(* IEC 61131-3 sources: POMIRTS_lab3/AS/Library_2/AsHydCon/V3.00.0, 3 files *)

(* ---- AsHydCon.typ ---- *)
TYPE
	HCRMovePara_typ : STRUCT
		t_Jolt	: REAL ;
		vC_pos	: REAL ;
		vC_neg	: REAL ;
		aAcc_pos	: REAL ;
		aDec_pos	: REAL ;
		aAcc_neg	: REAL ;
		aDec_neg	: REAL ;
	END_STRUCT;
	HCRSFG_Internal_typ : STRUCT
		SFG_Para	: HCRMovePara_typ ;
		Profile_Case	: USINT ;
		Fp_delta	: REAL ;
		Fp_brake	: REAL ;
		Fp_set_0	: REAL ;
		dFp_set_0	: REAL ;
		dFp_home	: REAL ;
		dFp_0_intrude	: USINT ;
		dFp_const	: REAL ;
		dFp_const_avg	: REAL ;
		dFp_thresh	: ARRAY[0..2] OF REAL ;
		t_Jolt	: REAL ;
		t_delta	: REAL ;
		t_delta_Jolt	: REAL ;
		t_delta_3_Jolt	: REAL ;
		Calc_t_delta	: USINT ;
		tx	: REAL ;
		tx_limit	: REAL ;
		enable_old	: BOOL ;
		Bootkey	: UDINT ;
	END_STRUCT;
	HCRF_Cont_InVar_typ : STRUCT
		I_Switch	: USINT ;
		Q_man	: REAL ;
		Q_add	: REAL ;
		v_act	: REAL ;
		Qy_Oset_ext	: REAL ;
		Oset_Mode	: USINT ;
	END_STRUCT;
	HCRP2P_Cont_Internal_typ : STRUCT
		MoveDir	: SINT ;
		s_set_old	: REAL ;
		enable_old	: BOOL ;
		Bootkey	: UDINT ;
	END_STRUCT;
	HCRP2P_Cont_AddPar_typ : STRUCT
		Y_P2P_min	: REAL ;
		Y_P2P_max	: REAL ;
		dY_max	: REAL ;
		Tn_pos	: REAL ;
		Tn_neg	: REAL ;
		I_Switch	: USINT ;
		Tv	: REAL ;
		Tf	: REAL ;
	END_STRUCT;
	HCRF_Cont_p_Internal_typ : STRUCT
		Qnom_pos	: REAL ;
		Qnom_neg	: REAL ;
		Oset_Mode	: USINT ;
		Qy_Oset_F_pos	: REAL ;
		Qy_Oset_F_neg	: REAL ;
		enable_old	: BOOL ;
		Bootkey	: UDINT ;
	END_STRUCT;
	HCRFyServo_Internal_typ : STRUCT
		E	: REAL ;
		Alpha	: REAL ;
		pSupply_max	: REAL ;
		pSupply	: REAL ;
		pTank	: REAL ;
		Qnom_pos	: REAL ;
		Qnom_neg	: REAL ;
		A_Cyl_pos	: REAL ;
		A_Cyl_neg	: REAL ;
		V0_pos	: REAL ;
		V0_neg	: REAL ;
		Neg_y	: BOOL ;
		dF_Cyl_sup	: REAL ;
		dF_Cyl_sum	: REAL ;
		x_Cyl	: REAL ;
		h_Cyl	: REAL ;
		h_Cyl_dbl_1	: UDINT ;
		h_Cyl_dbl_2	: UDINT ;
		K_pos_dbl_1	: UDINT ;
		K_pos_dbl_2	: UDINT ;
		K_neg_dbl_1	: UDINT ;
		K_neg_dbl_2	: UDINT ;
		V0_A_Cyl_pos_dbl_1	: UDINT ;
		V0_A_Cyl_pos_dbl_2	: UDINT ;
		V0_A_Cyl_neg_dbl_1	: UDINT ;
		V0_A_Cyl_neg_dbl_2	: UDINT ;
		A_Cyl_pos_1000_dbl_1	: UDINT ;
		A_Cyl_pos_1000_dbl_2	: UDINT ;
		A_Cyl_neg_1000_dbl_1	: UDINT ;
		A_Cyl_neg_1000_dbl_2	: UDINT ;
		E_10_dbl_1	: UDINT ;
		E_10_dbl_2	: UDINT ;
		pDelta_min_dbl_1	: UDINT ;
		pDelta_min_dbl_2	: UDINT ;
		dF_Cyl_sup_100_dbl_1	: UDINT ;
		dF_Cyl_sup_100_dbl_2	: UDINT ;
		Update_old	: USINT ;
		Update_2	: USINT ;
		enable_old	: BOOL ;
		Bootkey	: UDINT ;
	END_STRUCT;
	HCRNotch_Internal_typ : STRUCT
		Ts	: DINT ;
		Ts_dbl_1	: UDINT ;
		Ts_dbl_2	: UDINT ;
		fs_dbl_1	: UDINT ;
		fs_dbl_2	: UDINT ;
		V_old	: REAL ;
		f0_old	: REAL ;
		B_old	: REAL ;
		Set_y_old	: USINT ;
		Set_y_2	: USINT ;
		fg_upper	: REAL ;
		fg_lower	: REAL ;
		B_act	: REAL ;
		D	: REAL ;
		Tf	: REAL ;
		x1_dbl_1	: UDINT ;
		x1_dbl_2	: UDINT ;
		x2_dbl_1	: UDINT ;
		x2_dbl_2	: UDINT ;
		D_Ts_Tf_dbl_1	: UDINT ;
		D_Ts_Tf_dbl_2	: UDINT ;
		Sqrt_D_1_dbl_1	: UDINT ;
		Sqrt_D_1_dbl_2	: UDINT ;
		a0_dbl_1	: UDINT ;
		a0_dbl_2	: UDINT ;
		a1_dbl_1	: UDINT ;
		a1_dbl_2	: UDINT ;
		b0_dbl_1	: UDINT ;
		b0_dbl_2	: UDINT ;
		b1_dbl_1	: UDINT ;
		b1_dbl_2	: UDINT ;
		Bootkey	: UDINT ;
	END_STRUCT;
	HCRIT1_Internal_typ : STRUCT
		Ts	: DINT ;
		Ts_dbl_1	: UDINT ;
		Ts_dbl_2	: UDINT ;
		V_old	: REAL ;
		Tn_old	: REAL ;
		T1_old	: REAL ;
		Set_y_old	: USINT ;
		Set_y_2	: USINT ;
		x1_dbl_1	: UDINT ;
		x1_dbl_2	: UDINT ;
		x2_dbl_1	: UDINT ;
		x2_dbl_2	: UDINT ;
		Exp_Ts_T1_dbl_1	: UDINT ;
		Exp_Ts_T1_dbl_2	: UDINT ;
		V_Tn_dbl_1	: UDINT ;
		V_Tn_dbl_2	: UDINT ;
		a0_dbl_1	: UDINT ;
		a0_dbl_2	: UDINT ;
		a1_dbl_1	: UDINT ;
		a1_dbl_2	: UDINT ;
		b0_dbl_1	: UDINT ;
		b0_dbl_2	: UDINT ;
		b1_dbl_1	: UDINT ;
		b1_dbl_2	: UDINT ;
		Bootkey	: UDINT ;
	END_STRUCT;
	HCRSystemParaAdd_typ : STRUCT
		V0_pos	: REAL ;
		V0_neg	: REAL ;
		h_Cyl	: REAL ;
		m_Cyl	: REAL ;
	END_STRUCT;
	HCRRampGen_Internal_typ : STRUCT
		t_rise	: REAL ;
		t_hold	: REAL ;
		t_fall	: REAL ;
		y	: REAL ;
		dy	: REAL ;
		Finished	: BOOL ;
		Ts	: DINT ;
		Ts_dbl_1	: UDINT ;
		Ts_dbl_2	: UDINT ;
		Timer_dbl_1	: UDINT ;
		Timer_dbl_2	: UDINT ;
		k_Ramp_dbl_1	: UDINT ;
		k_Ramp_dbl_2	: UDINT ;
		y_dbl_1	: UDINT ;
		y_dbl_2	: UDINT ;
		RampGenPhase	: USINT ;
		enable_old	: BOOL ;
		Bootkey	: UDINT ;
	END_STRUCT;
	HCRAutoTune_Internal_typ : STRUCT
		E	: REAL ;
		V0_pos	: REAL ;
		V0_pos_mod_dbl_1	: UDINT ;
		V0_pos_mod_dbl_2	: UDINT ;
		V0_neg	: REAL ;
		V0_neg_mod_dbl_1	: UDINT ;
		V0_neg_mod_dbl_2	: UDINT ;
		s_Cyl_min_dbl_1	: UDINT ;
		s_Cyl_min_dbl_2	: UDINT ;
		s_Cyl_max_dbl_1	: UDINT ;
		s_Cyl_max_dbl_2	: UDINT ;
		h_Cyl	: REAL ;
		h_Cyl_dbl_1	: UDINT ;
		h_Cyl_dbl_2	: UDINT ;
		E_A_pos_2_dbl_1	: UDINT ;
		E_A_pos_2_dbl_2	: UDINT ;
		E_A_neg_2_dbl_1	: UDINT ;
		E_A_neg_2_dbl_2	: UDINT ;
		s0_Cyl	: REAL ;
		s0_Cyl_dbl_1	: UDINT ;
		s0_Cyl_dbl_2	: UDINT ;
		c0_Cyl	: REAL ;
		c0_Cyl_dbl_1	: UDINT ;
		c0_Cyl_dbl_2	: UDINT ;
		omega0_Cyl	: REAL ;
		omega0_Cyl_dbl_1	: UDINT ;
		omega0_Cyl_dbl_2	: UDINT ;
		vCyl_sup_pos	: REAL ;
		vCyl_sup_neg	: REAL ;
		vCyl_sup	: REAL ;
		Kp_dbl_1	: UDINT ;
		Kp_dbl_2	: UDINT ;
		Kp_physical	: REAL ;
		enable_old	: BOOL ;
		Bootkey	: UDINT ;
	END_STRUCT;
	HCRs_Cont_p_InVar_typ : STRUCT
		I_Switch	: USINT ;
		v_man	: REAL ;
		v_add	: REAL ;
		v_set	: REAL ;
		pCyl_pos	: REAL ;
		pCyl_neg	: REAL ;
		Qy_Oset_ext	: REAL ;
		Oset_Mode	: USINT ;
	END_STRUCT;
	HCRsF_Cont_p_Internal_typ : STRUCT
		CTRLmode	: USINT ;
		uSwitch_old	: USINT ;
		enable_old	: BOOL ;
		Bootkey	: UDINT ;
	END_STRUCT;
	HCRs_Cont_p_Internal_typ : STRUCT
		vCyl_sup_pos	: REAL ;
		vCyl_sup_neg	: REAL ;
		vCyl_sup	: REAL ;
		s_set_old	: REAL ;
		s_act_old	: REAL ;
		v_act	: REAL ;
		Oset_Mode	: USINT ;
		Qy_Oset_s_pos	: REAL ;
		Qy_Oset_s_neg	: REAL ;
		Qy_I_Switch	: USINT ;
		Qy_I	: REAL ;
		MoveDir_I	: SINT ;
		enable_old	: BOOL ;
		Bootkey	: UDINT ;
	END_STRUCT;
	HCROmega0_Internal_typ : STRUCT
		E	: REAL ;
		Kp_xCorr_Lim	: REAL ;
		A_Cyl_pos	: REAL ;
		A_Cyl_neg	: REAL ;
		V0_pos	: REAL ;
		V0_neg	: REAL ;
		h_Cyl	: REAL ;
		x_Cyl_min_dbl_1	: UDINT ;
		x_Cyl_min_dbl_2	: UDINT ;
		x_Cyl_max_dbl_1	: UDINT ;
		x_Cyl_max_dbl_2	: UDINT ;
		E_A_pos_2_dbl_1	: UDINT ;
		E_A_pos_2_dbl_2	: UDINT ;
		E_A_neg_2_dbl_1	: UDINT ;
		E_A_neg_2_dbl_2	: UDINT ;
		x0_Cyl_dbl_1	: UDINT ;
		x0_Cyl_dbl_2	: UDINT ;
		c0_Cyl	: REAL ;
		c0_Cyl_dbl_1	: UDINT ;
		c0_Cyl_dbl_2	: UDINT ;
		c_Cyl_Lim_L	: REAL ;
		c_Cyl_Lim_L_dbl_1	: UDINT ;
		c_Cyl_Lim_L_dbl_2	: UDINT ;
		c_Cyl_Lim_R	: REAL ;
		c_Cyl_Lim_R_dbl_1	: UDINT ;
		c_Cyl_Lim_R_dbl_2	: UDINT ;
		c_Cyl	: REAL ;
		c_Cyl_dbl_1	: UDINT ;
		c_Cyl_dbl_2	: UDINT ;
		Kp_xCorr_Lim_L	: REAL ;
		Kp_xCorr_Lim_R	: REAL ;
		enable_old	: BOOL ;
		Bootkey	: UDINT ;
	END_STRUCT;
	HCRLinValve_Internal_typ : STRUCT
		Neg_Uy	: BOOL ;
		enable_old	: BOOL ;
		Bootkey	: UDINT ;
	END_STRUCT;
	HCRFIFO_Internal_typ : STRUCT
		Ts	: DINT ;
		t_FIFO_max	: DINT ;
		MemSize	: UDINT ;
		MemSize_REAL	: UDINT ;
		Set_y_2	: BOOL ;
		pFIFO_Buf	: UDINT ;
		pFIFO_OutIn	: UDINT ;
		enable_old	: BOOL ;
		Bootkey	: UDINT ;
	END_STRUCT;
	HCRDT2_Internal_typ : STRUCT
		Ts	: DINT ;
		Ts_dbl_1	: UDINT ;
		Ts_dbl_2	: UDINT ;
		Tv_old	: REAL ;
		T1_old	: REAL ;
		T2_old	: REAL ;
		n_Avg_old	: USINT ;
		u_Buf	: ARRAY[0..99] OF REAL ;
		u_BufCnt	: SINT ;
		u_Sum_dbl_1	: UDINT ;
		u_Sum_dbl_2	: UDINT ;
		u_Avg_dbl_1	: UDINT ;
		u_Avg_dbl_2	: UDINT ;
		Reset_y_old	: USINT ;
		Reset_y_2	: USINT ;
		x1_dbl_1	: UDINT ;
		x1_dbl_2	: UDINT ;
		x2_dbl_1	: UDINT ;
		x2_dbl_2	: UDINT ;
		Tv_T1_dbl_1	: UDINT ;
		Tv_T1_dbl_2	: UDINT ;
		Tv_T2_dbl_1	: UDINT ;
		Tv_T2_dbl_2	: UDINT ;
		Exp_Ts_T1_dbl_1	: UDINT ;
		Exp_Ts_T1_dbl_2	: UDINT ;
		Exp_Ts_T2_dbl_1	: UDINT ;
		Exp_Ts_T2_dbl_2	: UDINT ;
		Exp_T1_T2_dbl_1	: UDINT ;
		Exp_T1_T2_dbl_2	: UDINT ;
		a0_dbl_1	: UDINT ;
		a0_dbl_2	: UDINT ;
		a1_dbl_1	: UDINT ;
		a1_dbl_2	: UDINT ;
		b0_dbl_1	: UDINT ;
		b0_dbl_2	: UDINT ;
		b1_dbl_1	: UDINT ;
		b1_dbl_2	: UDINT ;
		Bootkey	: UDINT ;
	END_STRUCT;
	HCRF_Cont_p_InVar_typ : STRUCT
		I_Switch	: USINT ;
		Q_man	: REAL ;
		Q_add	: REAL ;
		dFp_set	: REAL ;
		x_Cyl	: REAL ;
		v_Cyl	: REAL ;
		pCyl_pos	: REAL ;
		pCyl_neg	: REAL ;
		v_act	: REAL ;
		Qy_Oset_ext	: REAL ;
		Oset_Mode	: USINT ;
	END_STRUCT;
	HCRs_Cont_InVar_typ : STRUCT
		I_Switch	: USINT ;
		v_man	: REAL ;
		v_add	: REAL ;
		v_set	: REAL ;
		Fp_Cyl	: REAL ;
		Ff_Cyl_pos	: REAL ;
		Ff_Cyl_neg	: REAL ;
		Qy_Oset_ext	: REAL ;
		Oset_Mode	: USINT ;
	END_STRUCT;
	HCRsF_Cont_Internal_typ : STRUCT
		uSwitch_old	: USINT ;
		enable_old	: BOOL ;
		Bootkey	: UDINT ;
	END_STRUCT;
	HCRPIDPara_F_typ : STRUCT
		Fp_min	: REAL ;
		Fp_max	: REAL ;
		Kw	: REAL ;
		Kp	: REAL ;
		Tn	: REAL ;
		K_Fbk	: REAL ;
		d_mode	: USINT ;
		Tv	: REAL ;
		Tf	: REAL ;
		dQ_max	: REAL ;
		Q_min	: REAL ;
		Q_max	: REAL ;
	END_STRUCT;
	HCRPIDPara_s_typ : STRUCT
		s_min	: REAL ;
		s_max	: REAL ;
		Kw	: REAL ;
		Kp	: REAL ;
		Tn_pos	: REAL ;
		Tn_neg	: REAL ;
		K_Fbk	: REAL ;
		d_mode	: USINT ;
		Tv	: REAL ;
		Tf	: REAL ;
		dv_max	: REAL ;
		v_min	: REAL ;
		v_max	: REAL ;
	END_STRUCT;
	HCRF_Cont_Internal_typ : STRUCT
		Qnom_pos	: REAL ;
		Qnom_neg	: REAL ;
		Oset_Mode	: USINT ;
		Qy_Oset_F_pos	: REAL ;
		Qy_Oset_F_neg	: REAL ;
		enable_old	: BOOL ;
		Bootkey	: UDINT ;
	END_STRUCT;
	HCRJoltFree_Internal_typ : STRUCT
		uSwitch_old	: BOOL ;
		enable_old	: BOOL ;
		Bootkey	: UDINT ;
	END_STRUCT;
	HCRDT2s_Internal_typ : STRUCT
		Ts	: DINT ;
		Ts_dbl_1	: UDINT ;
		Ts_dbl_2	: UDINT ;
		D_old	: REAL ;
		Tv_old	: REAL ;
		Tf_old	: REAL ;
		Reset_y_old	: USINT ;
		Reset_y_2	: USINT ;
		x1_dbl_1	: UDINT ;
		x1_dbl_2	: UDINT ;
		x2_dbl_1	: UDINT ;
		x2_dbl_2	: UDINT ;
		Sqrt_D_1_dbl_1	: UDINT ;
		Sqrt_D_1_dbl_2	: UDINT ;
		Tv_Tf_dbl_1	: UDINT ;
		Tv_Tf_dbl_2	: UDINT ;
		Ts_Tf_dbl_1	: UDINT ;
		Ts_Tf_dbl_2	: UDINT ;
		Exp_D_Ts_Tf_dbl_1	: UDINT ;
		Exp_D_Ts_Tf_dbl_2	: UDINT ;
		a0_dbl_1	: UDINT ;
		a0_dbl_2	: UDINT ;
		a1_dbl_1	: UDINT ;
		a1_dbl_2	: UDINT ;
		b0_dbl_1	: UDINT ;
		b0_dbl_2	: UDINT ;
		b1_dbl_1	: UDINT ;
		b1_dbl_2	: UDINT ;
		Bootkey	: UDINT ;
	END_STRUCT;
	HCRPT1cP_Internal_typ : STRUCT
		Ts	: DINT ;
		Ts_dbl_1	: UDINT ;
		Ts_dbl_2	: UDINT ;
		T1_intern	: REAL ;
		nCnt	: UDINT ;
		Set_y_old	: USINT ;
		Set_y_2	: USINT ;
		x_dbl_1	: UDINT ;
		x_dbl_2	: UDINT ;
		Exp_5_dbl_1	: UDINT ;
		Exp_5_dbl_2	: UDINT ;
		a0_dbl_1	: UDINT ;
		a0_dbl_2	: UDINT ;
		b0_dbl_1	: UDINT ;
		b0_dbl_2	: UDINT ;
		Bootkey	: UDINT ;
	END_STRUCT;
	HCRPT2s_Internal_typ : STRUCT
		Ts	: DINT ;
		Ts_dbl_1	: UDINT ;
		Ts_dbl_2	: UDINT ;
		V_old	: REAL ;
		D_old	: REAL ;
		Tf_old	: REAL ;
		Set_y_old	: USINT ;
		Set_y_2	: USINT ;
		x1_dbl_1	: UDINT ;
		x1_dbl_2	: UDINT ;
		x2_dbl_1	: UDINT ;
		x2_dbl_2	: UDINT ;
		Sqrt_D_1_dbl_1	: UDINT ;
		Sqrt_D_1_dbl_2	: UDINT ;
		Ts_Tf_dbl_1	: UDINT ;
		Ts_Tf_dbl_2	: UDINT ;
		Exp_D_Ts_Tf_dbl_1	: UDINT ;
		Exp_D_Ts_Tf_dbl_2	: UDINT ;
		a0_dbl_1	: UDINT ;
		a0_dbl_2	: UDINT ;
		a1_dbl_1	: UDINT ;
		a1_dbl_2	: UDINT ;
		b0_dbl_1	: UDINT ;
		b0_dbl_2	: UDINT ;
		b1_dbl_1	: UDINT ;
		b1_dbl_2	: UDINT ;
		Bootkey	: UDINT ;
	END_STRUCT;
	HCRPT2_Internal_typ : STRUCT
		Ts	: DINT ;
		Ts_dbl_1	: UDINT ;
		Ts_dbl_2	: UDINT ;
		V_old	: REAL ;
		T1_old	: REAL ;
		T2_old	: REAL ;
		Set_y_old	: USINT ;
		Set_y_2	: USINT ;
		x1_dbl_1	: UDINT ;
		x1_dbl_2	: UDINT ;
		x2_dbl_1	: UDINT ;
		x2_dbl_2	: UDINT ;
		Exp_Ts_T1_dbl_1	: UDINT ;
		Exp_Ts_T1_dbl_2	: UDINT ;
		Exp_Ts_T2_dbl_1	: UDINT ;
		Exp_Ts_T2_dbl_2	: UDINT ;
		Exp_Ts_T1_T2_dbl_1	: UDINT ;
		Exp_Ts_T1_T2_dbl_2	: UDINT ;
		Exp_T1_T2_dbl_1	: UDINT ;
		Exp_T1_T2_dbl_2	: UDINT ;
		V1_Exp_dbl_1	: UDINT ;
		V1_Exp_dbl_2	: UDINT ;
		V2_Exp_dbl_1	: UDINT ;
		V2_Exp_dbl_2	: UDINT ;
		Bootkey	: UDINT ;
	END_STRUCT;
	HCRPT1_Internal_typ : STRUCT
		Ts	: DINT ;
		Ts_dbl_1	: UDINT ;
		Ts_dbl_2	: UDINT ;
		V_old	: REAL ;
		T1_old	: REAL ;
		Set_y_old	: USINT ;
		Set_y_2	: USINT ;
		x_dbl_1	: UDINT ;
		x_dbl_2	: UDINT ;
		Exp_Ts_T1_dbl_1	: UDINT ;
		Exp_Ts_T1_dbl_2	: UDINT ;
		V_Exp_dbl_1	: UDINT ;
		V_Exp_dbl_2	: UDINT ;
		Bootkey	: UDINT ;
	END_STRUCT;
	HCRDT1_Internal_typ : STRUCT
		Ts	: DINT ;
		Ts_dbl_1	: UDINT ;
		Ts_dbl_2	: UDINT ;
		Tv_old	: REAL ;
		Tf_old	: REAL ;
		n_Avg_old	: USINT ;
		u_Buf	: ARRAY[0..99] OF REAL ;
		u_BufCnt	: SINT ;
		u_Sum_dbl_1	: UDINT ;
		u_Sum_dbl_2	: UDINT ;
		u_Avg_dbl_1	: UDINT ;
		u_Avg_dbl_2	: UDINT ;
		Reset_y_old	: USINT ;
		Reset_y_2	: USINT ;
		x_dbl_1	: UDINT ;
		x_dbl_2	: UDINT ;
		Tv_Tf_dbl_1	: UDINT ;
		Tv_Tf_dbl_2	: UDINT ;
		Exp_Ts_Tf_dbl_1	: UDINT ;
		Exp_Ts_Tf_dbl_2	: UDINT ;
		Tv_Tf_Exp_dbl_1	: UDINT ;
		Tv_Tf_Exp_dbl_2	: UDINT ;
		V_Exp_dbl_1	: UDINT ;
		V_Exp_dbl_2	: UDINT ;
		Bootkey	: UDINT ;
	END_STRUCT;
	HCRFyServo_Fp_Internal_typ : STRUCT
		Alpha	: REAL ;
		pSupply_max	: REAL ;
		pSupply	: REAL ;
		pTank	: REAL ;
		Qnom_pos	: REAL ;
		Qnom_neg	: REAL ;
		A_Cyl_pos	: REAL ;
		A_Cyl_neg	: REAL ;
		Neg_y	: BOOL ;
		Supply_Tank_pos_dbl_1	: UDINT ;
		Supply_Tank_pos_dbl_2	: UDINT ;
		Supply_Tank_neg_dbl_1	: UDINT ;
		Supply_Tank_neg_dbl_2	: UDINT ;
		K_numer_dbl_1	: UDINT ;
		K_numer_dbl_2	: UDINT ;
		Update_old	: USINT ;
		Update_2	: USINT ;
		enable_old	: BOOL ;
		Bootkey	: UDINT ;
	END_STRUCT;
	HCRSPF_Internal_typ : STRUCT
		Profile_Nb	: USINT ;
		Profile_ID	: USINT ;
		Profile_Case	: USINT ;
		MovementPhase	: USINT ;
		MovementStep	: USINT ;
		s_end	: REAL ;
		s_set_0_dbl_1	: UDINT ;
		s_set_0_dbl_2	: UDINT ;
		v_set_0_dbl_1	: UDINT ;
		v_set_0_dbl_2	: UDINT ;
		a_set_0_dbl_1	: UDINT ;
		a_set_0_dbl_2	: UDINT ;
		v0	: REAL ;
		v0_dbl_1	: UDINT ;
		v0_dbl_2	: UDINT ;
		v0_intrude	: USINT ;
		v0_state	: USINT ;
		s_set	: REAL ;
		s_set_Jolt	: REAL ;
		s_set_dbl_1	: UDINT ;
		s_set_dbl_2	: UDINT ;
		v_set	: REAL ;
		v_set_Jolt	: REAL ;
		v_set_dbl_1	: UDINT ;
		v_set_dbl_2	: UDINT ;
		a_set	: REAL ;
		a_set_Jolt	: REAL ;
		a_set_dbl_1	: UDINT ;
		a_set_dbl_2	: UDINT ;
		vC_pos_dbl_1	: UDINT ;
		vC_pos_dbl_2	: UDINT ;
		vC_neg_dbl_1	: UDINT ;
		vC_neg_dbl_2	: UDINT ;
		aAcc_pos_dbl_1	: UDINT ;
		aAcc_pos_dbl_2	: UDINT ;
		aDec_pos_dbl_1	: UDINT ;
		aDec_pos_dbl_2	: UDINT ;
		aAcc_neg_dbl_1	: UDINT ;
		aAcc_neg_dbl_2	: UDINT ;
		aDec_neg_dbl_1	: UDINT ;
		aDec_neg_dbl_2	: UDINT ;
		aDec	: REAL ;
		aDec_intrude	: BOOL ;
		s_period	: REAL ;
		s_period_Sum_dbl_1	: UDINT ;
		s_period_Sum_dbl_2	: UDINT ;
		Nb_period	: DINT ;
		t_Jolt_max	: REAL ;
		t_Jolt_limit	: REAL ;
		t_Jolt	: REAL ;
		t_Jolt_dbl_1	: UDINT ;
		t_Jolt_dbl_2	: UDINT ;
		sDelta	: REAL ;
		sDelta_dbl_1	: UDINT ;
		sDelta_dbl_2	: UDINT ;
		sBrake	: REAL ;
		sBrake_dbl_1	: UDINT ;
		sBrake_dbl_2	: UDINT ;
		vTop	: REAL ;
		vTop_dbl_1	: UDINT ;
		vTop_dbl_2	: UDINT ;
		AccVec_dbl	: ARRAY[0..39] OF UDINT ;
		ConstVec_dbl	: ARRAY[0..39] OF UDINT ;
		DecVec_dbl	: ARRAY[0..39] OF UDINT ;
		AccVec	: ARRAY[0..19] OF REAL ;
		ConstVec	: ARRAY[0..19] OF REAL ;
		DecVec	: ARRAY[0..19] OF REAL ;
		pBuf_s_set	: UDINT ;
		pBuf_v_set	: UDINT ;
		pBuf_a_set	: UDINT ;
		BufCntMax	: DINT ;
		BufCnt	: DINT ;
		BufCnt_t_Jolt	: DINT ;
		Cnt_t_Jolt	: DINT ;
		s_set_Sum_dbl_1	: UDINT ;
		s_set_Sum_dbl_2	: UDINT ;
		D	: REAL ;
		omega0	: REAL ;
		t_pred	: REAL ;
		Ts	: DINT ;
		Ts_dbl_1	: UDINT ;
		Ts_dbl_2	: UDINT ;
		Ts_2_dbl_1	: UDINT ;
		Ts_2_dbl_2	: UDINT ;
		Ts_4_dbl_1	: UDINT ;
		Ts_4_dbl_2	: UDINT ;
		Timer	: REAL ;
		Timer_dbl_1	: UDINT ;
		Timer_dbl_2	: UDINT ;
		Timer_Ts	: REAL ;
		Timer_Ts_dbl_1	: UDINT ;
		Timer_Ts_dbl_2	: UDINT ;
		T_cycle	: REAL ;
		T_cycle_dbl_1	: UDINT ;
		T_cycle_dbl_2	: UDINT ;
		Const_T_cycle	: BOOL ;
		CounterState	: UINT ;
		musecs_old	: UDINT ;
		SysTicks_old	: UDINT ;
		enable_old	: BOOL ;
		Bootkey_T	: UDINT ;
		Bootkey	: UDINT ;
		s_period_ext	: REAL ;
		PeriodicMode_ext	: INT ;
		NewPeriod_ext_out	: SINT ;
	END_STRUCT;
	HCRs_Cont_Internal_typ : STRUCT
		vCyl_sup_pos	: REAL ;
		vCyl_sup_neg	: REAL ;
		vCyl_sup	: REAL ;
		s_set_old	: REAL ;
		s_act_old	: REAL ;
		v_act	: REAL ;
		Oset_Mode	: USINT ;
		Qy_Oset_s_pos	: REAL ;
		Qy_Oset_s_neg	: REAL ;
		Qy_I_Switch	: USINT ;
		Qy_I	: REAL ;
		MoveDir_I	: SINT ;
		enable_old	: BOOL ;
		Bootkey	: UDINT ;
	END_STRUCT;
	HCRSystemPara_typ : STRUCT
		pSupply_max	: REAL ;
		pSupply	: REAL ;
		pTank	: REAL ;
		A_Cyl_pos	: REAL ;
		A_Cyl_neg	: REAL ;
	END_STRUCT;
	HCRValvePara_typ : STRUCT
		Qnom_pos	: REAL ;
		Qnom_neg	: REAL ;
		pDelta_nom	: REAL ;
		yValve_0	: REAL ;
		Neg_y	: BOOL ;
	END_STRUCT;
	HCRPIDPara_typ : STRUCT
		WX_min	: REAL ;
		WX_max	: REAL ;
		Kw	: REAL ;
		Kp	: REAL ;
		Tn_pos	: REAL ;
		Tn_neg	: REAL ;
		K_Fbk	: REAL ;
		d_mode	: USINT ;
		Tv	: REAL ;
		Tf	: REAL ;
		dY_max	: REAL ;
		Y_min	: REAL ;
		Y_max	: REAL ;
	END_STRUCT;
	HCRPID_Internal_typ : STRUCT
		WX_min	: REAL ;
		WX_max	: REAL ;
		_100_WX_delta_dbl_1	: UDINT ;
		_100_WX_delta_dbl_2	: UDINT ;
		W_norm_dbl_1	: UDINT ;
		W_norm_dbl_2	: UDINT ;
		X_norm_dbl_1	: UDINT ;
		X_norm_dbl_2	: UDINT ;
		Invert	: BOOL ;
		e_norm_dbl_1	: UDINT ;
		e_norm_dbl_2	: UDINT ;
		Kp	: REAL ;
		Kw	: REAL ;
		Kp_Kw_1_dbl_1	: UDINT ;
		Kp_Kw_1_dbl_2	: UDINT ;
		Kp_intrude	: REAL ;
		P_intrude	: BOOL ;
		Yp_dbl_1	: UDINT ;
		Yp_dbl_2	: UDINT ;
		Ts	: DINT ;
		Ts_dbl_1	: UDINT ;
		Ts_dbl_2	: UDINT ;
		Tn_pos_dbl_1	: UDINT ;
		Tn_pos_dbl_2	: UDINT ;
		Tn_neg_dbl_1	: UDINT ;
		Tn_neg_dbl_2	: UDINT ;
		Kp_Ts_Tn_pos_dbl_1	: UDINT ;
		Kp_Ts_Tn_pos_dbl_2	: UDINT ;
		Kp_Ts_Tn_neg_dbl_1	: UDINT ;
		Kp_Ts_Tn_neg_dbl_2	: UDINT ;
		Yi_load	: REAL ;
		I_load	: SINT ;
		Yi_dbl_1	: UDINT ;
		Yi_dbl_2	: UDINT ;
		Yi_pos_last_dbl_1	: UDINT ;
		Yi_pos_last_dbl_2	: UDINT ;
		Yi_neg_last_dbl_1	: UDINT ;
		Yi_neg_last_dbl_2	: UDINT ;
		I_Switch_Sign	: SINT ;
		I_Switch	: SINT ;
		I_Switch_old	: SINT ;
		I_Switch_off	: SINT ;
		d_mode	: USINT ;
		D	: REAL ;
		Tv_dbl_1	: UDINT ;
		Tv_dbl_2	: UDINT ;
		Tf_dbl_1	: UDINT ;
		Tf_dbl_2	: UDINT ;
		x1d_dbl_1	: UDINT ;
		x1d_dbl_2	: UDINT ;
		x2d_dbl_1	: UDINT ;
		x2d_dbl_2	: UDINT ;
		a0d_dbl_1	: UDINT ;
		a0d_dbl_2	: UDINT ;
		a1d_dbl_1	: UDINT ;
		a1d_dbl_2	: UDINT ;
		b0d_dbl_1	: UDINT ;
		b0d_dbl_2	: UDINT ;
		b1d_dbl_1	: UDINT ;
		b1d_dbl_2	: UDINT ;
		Yd_dbl_1	: UDINT ;
		Yd_dbl_2	: UDINT ;
		Reset_Yd	: USINT ;
		Y_min	: REAL ;
		Y_max	: REAL ;
		Ytotal_dbl_1	: UDINT ;
		Ytotal_dbl_2	: UDINT ;
		Ylim_dbl_1	: UDINT ;
		Ylim_dbl_2	: UDINT ;
		Y_Fbk_ext	: REAL ;
		Fbk_mode	: USINT ;
		K_Fbk_Kp_dbl_1	: UDINT ;
		K_Fbk_Kp_dbl_2	: UDINT ;
		e_Fbk_dbl_1	: UDINT ;
		e_Fbk_dbl_2	: UDINT ;
		dY_max	: REAL ;
		dY_max_Ts_dbl_1	: UDINT ;
		dY_max_Ts_dbl_2	: UDINT ;
		Y_dbl_1	: UDINT ;
		Y_dbl_2	: UDINT ;
		UpdateValid	: BOOL ;
		enable_old	: BOOL ;
		Bootkey_CM	: UDINT ;
		Bootkey	: UDINT ;
	END_STRUCT;
	HCRvyServo_Internal_typ : STRUCT
		Alpha	: REAL ;
		vCyl_sup_pos	: REAL ;
		vCyl_sup_neg	: REAL ;
		vCyl_sup	: REAL ;
		vCyl_max_pos	: REAL ;
		vCyl_max_neg	: REAL ;
		vCyl_max	: REAL ;
		vCyl_sum	: REAL ;
		vCyl_thresh	: REAL ;
		vCyl_nOverlap_pos	: REAL ;
		vCyl_nOverlap_neg	: REAL ;
		vCyl_old	: REAL ;
		pSupply_max	: REAL ;
		pSupply	: REAL ;
		pTank	: REAL ;
		Qnom_pos	: REAL ;
		Qnom_neg	: REAL ;
		A_Cyl_pos	: REAL ;
		A_Cyl_neg	: REAL ;
		yValve_zero	: REAL ;
		yValve_min	: REAL ;
		Neg_y	: BOOL ;
		yValve_0	: REAL ;
		yValve_0_dbl_1	: UDINT ;
		yValve_0_dbl_2	: UDINT ;
		K_pos_dbl_1	: UDINT ;
		K_pos_dbl_2	: UDINT ;
		K_neg_dbl_1	: UDINT ;
		K_neg_dbl_2	: UDINT ;
		K_nOverlap_pos_dbl_1	: UDINT ;
		K_nOverlap_pos_dbl_2	: UDINT ;
		K_nOverlap_neg_dbl_1	: UDINT ;
		K_nOverlap_neg_dbl_2	: UDINT ;
		S_nOverlap_dbl_1	: UDINT ;
		S_nOverlap_dbl_2	: UDINT ;
		pDelta_min_dbl_1	: UDINT ;
		pDelta_min_dbl_2	: UDINT ;
		vCyl_sup_100_dbl_1	: UDINT ;
		vCyl_sup_100_dbl_2	: UDINT ;
		Update_old	: USINT ;
		Update_2	: USINT ;
		enable_old	: BOOL ;
		Bootkey	: UDINT ;
	END_STRUCT;
	HCRvyServo_Fp_Internal_typ : STRUCT
		Alpha	: REAL ;
		vCyl_sup_pos	: REAL ;
		vCyl_sup_neg	: REAL ;
		vCyl_sup	: REAL ;
		vCyl_max_pos	: REAL ;
		vCyl_max_neg	: REAL ;
		vCyl_max	: REAL ;
		vCyl_sum	: REAL ;
		vCyl_thresh	: REAL ;
		vCyl_nOverlap_pos	: REAL ;
		vCyl_nOverlap_neg	: REAL ;
		vCyl_old	: REAL ;
		pSupply_max	: REAL ;
		pSupply	: REAL ;
		pTank	: REAL ;
		Qnom_pos	: REAL ;
		Qnom_neg	: REAL ;
		A_Cyl_pos	: REAL ;
		A_Cyl_neg	: REAL ;
		pCyl_pos	: REAL ;
		pCyl_neg	: REAL ;
		yValve_zero	: REAL ;
		yValve_min	: REAL ;
		Neg_y	: BOOL ;
		yValve_0	: REAL ;
		yValve_0_dbl_1	: UDINT ;
		yValve_0_dbl_2	: UDINT ;
		Supply_Tank_pos_dbl_1	: UDINT ;
		Supply_Tank_pos_dbl_2	: UDINT ;
		Supply_Tank_neg_dbl_1	: UDINT ;
		Supply_Tank_neg_dbl_2	: UDINT ;
		Qn_pos_2_A_neg_2_dbl_1	: UDINT ;
		Qn_pos_2_A_neg_2_dbl_2	: UDINT ;
		Qn_neg_2_A_pos_2_dbl_1	: UDINT ;
		Qn_neg_2_A_pos_2_dbl_2	: UDINT ;
		Qn_pos_2_A_neg_3_dbl_1	: UDINT ;
		Qn_pos_2_A_neg_3_dbl_2	: UDINT ;
		Qn_neg_2_A_pos_3_dbl_1	: UDINT ;
		Qn_neg_2_A_pos_3_dbl_2	: UDINT ;
		K_dbl_1	: UDINT ;
		K_dbl_2	: UDINT ;
		K_pos_dbl_1	: UDINT ;
		K_pos_dbl_2	: UDINT ;
		K_neg_dbl_1	: UDINT ;
		K_neg_dbl_2	: UDINT ;
		K_nOverlap_dbl_1	: UDINT ;
		K_nOverlap_dbl_2	: UDINT ;
		K_nOverlap_pos_dbl_1	: UDINT ;
		K_nOverlap_pos_dbl_2	: UDINT ;
		K_nOverlap_neg_dbl_1	: UDINT ;
		K_nOverlap_neg_dbl_2	: UDINT ;
		S_nOverlap_dbl_1	: UDINT ;
		S_nOverlap_dbl_2	: UDINT ;
		pCyl_pos_Numer_pos_dbl_1	: UDINT ;
		pCyl_pos_Numer_pos_dbl_2	: UDINT ;
		pCyl_neg_Numer_pos_dbl_1	: UDINT ;
		pCyl_neg_Numer_pos_dbl_2	: UDINT ;
		pCyl_pos_Numer_neg_dbl_1	: UDINT ;
		pCyl_pos_Numer_neg_dbl_2	: UDINT ;
		pCyl_neg_Numer_neg_dbl_1	: UDINT ;
		pCyl_neg_Numer_neg_dbl_2	: UDINT ;
		pCyl_Denom_dbl_1	: UDINT ;
		pCyl_Denom_dbl_2	: UDINT ;
		vCyl_sup_100_dbl_1	: UDINT ;
		vCyl_sup_100_dbl_2	: UDINT ;
		Update_old	: USINT ;
		Update_2	: USINT ;
		enable_old	: BOOL ;
		Bootkey	: UDINT ;
	END_STRUCT;
	HCRLinSpline_Internal_typ : STRUCT
		AscendingX_o	: SINT ;
		AscendingXs_o	: SINT ;
		AscendingY_o	: SINT ;
		AscendingYs_o	: SINT ;
		AscendingX_d	: SINT ;
		AscendingXs_d	: SINT ;
		AscendingY_d	: SINT ;
		AscendingYs_d	: SINT ;
		Rness_crit	: REAL ;
		RnessP	: REAL ;
		RnessR	: REAL ;
		_Smooth1_dbl_1	: UDINT ;
		_Smooth1_dbl_2	: UDINT ;
		_1Smooth_dbl_1	: UDINT ;
		_1Smooth_dbl_2	: UDINT ;
		_1Smooth1_dbl_1	: UDINT ;
		_1Smooth1_dbl_2	: UDINT ;
		enable_old	: BOOL ;
		Bootkey	: UDINT ;
	END_STRUCT;
	HCRNode_Internal_typ : STRUCT
		X	: REAL ;
		Y	: REAL ;
		X1	: REAL ;
		X2	: REAL ;
		Rness_crit	: REAL ;
		X1_dbl_1	: UDINT ;
		X1_dbl_2	: UDINT ;
		X2_dbl_1	: UDINT ;
		X2_dbl_2	: UDINT ;
		deltaX_dbl_1	: UDINT ;
		deltaX_dbl_2	: UDINT ;
		deltaY_dbl_1	: UDINT ;
		deltaY_dbl_2	: UDINT ;
		k_dbl_1	: UDINT ;
		k_dbl_2	: UDINT ;
		d_dbl_1	: UDINT ;
		d_dbl_2	: UDINT ;
	END_STRUCT;
	HCRNode_typ : STRUCT
		X	: REAL ;
		Y	: REAL ;
		Internal	: HCRNode_Internal_typ ;
	END_STRUCT;
END_TYPE

(* ---- AsHydCon.fun ---- *)
FUNCTION_BLOCK HCRsF_Cont_p (* Switchable position/force controller (pressure). *)
	VAR_INPUT
		enable	:BOOL;
		pSystem_Para	:REFERENCE TO HCRSystemPara_typ;
		pSystem_ParaAdd	:REFERENCE TO HCRSystemParaAdd_typ;
		pValve_Para	:REFERENCE TO HCRValvePara_typ;
		pPID_Para_s	:REFERENCE TO HCRPIDPara_s_typ;
		pPID_Para_F	:REFERENCE TO HCRPIDPara_F_typ;
		vyServoMode	:USINT;
		FyServoMode	:USINT;
		tSwitch	:REAL;
		Update	:USINT;
		s_set	:REAL;
		s_act	:REAL;
		s_Cont_p_InVar	:HCRs_Cont_p_InVar_typ;
		Fp_set	:REAL;
		Fp_act	:REAL;
		F_Cont_InVar	:HCRF_Cont_p_InVar_typ;
		CTRLmode	:USINT;
		uSwitch	:USINT;
	END_VAR
	VAR_OUTPUT
		Qy_s	:REAL;
		Qy_Oset_s	:REAL;
		Qy_F	:REAL;
		Qy_Oset_F	:REAL;
		Qy	:REAL;
		yValve	:REAL;
		MoveDir	:SINT;
		status	:UINT;
	END_VAR
	VAR
		Internal	:HCRsF_Cont_p_Internal_typ;
		s_Cont_p	:HCRs_Cont_p;
		F_Cont	:HCRF_Cont;
		F_Cont_p	:HCRF_Cont_p;
		vyServo	:HCRvyServo;
		JoltFree	:HCRJoltFree;
	END_VAR
END_FUNCTION_BLOCK
FUNCTION_BLOCK HCRNotch (* 2nd order notch filter. *)
	VAR_INPUT
		enable	:BOOL;
		V	:REAL;
		f0	:REAL;
		B	:REAL;
		u	:REAL;
		Set_y	:USINT;
		y_set	:REAL;
	END_VAR
	VAR_OUTPUT
		y	:REAL;
		status	:UINT;
	END_VAR
	VAR
		Internal	:HCRNotch_Internal_typ;
	END_VAR
END_FUNCTION_BLOCK
FUNCTION_BLOCK HCRs_Cont_p (* Position controller (pressure). *)
	VAR_INPUT
		enable	:BOOL;
		pSystem_Para	:REFERENCE TO HCRSystemPara_typ;
		pValve_Para	:REFERENCE TO HCRValvePara_typ;
		pPID_Para_s	:REFERENCE TO HCRPIDPara_s_typ;
		vyServoMode	:USINT;
		Update	:USINT;
		s_set	:REAL;
		s_act	:REAL;
		Invert	:BOOL;
		I_Switch	:USINT;
		CTRLmode	:USINT;
		v_man	:REAL;
		v_add	:REAL;
		v_set	:REAL;
		pCyl_pos	:REAL;
		pCyl_neg	:REAL;
		Qy_Oset_ext	:REAL;
		Oset_Mode	:USINT;
	END_VAR
	VAR_OUTPUT
		Qy_s	:REAL;
		Qy_Oset_s	:REAL;
		Qy	:REAL;
		yValve	:REAL;
		MoveDir	:SINT;
		status	:UINT;
	END_VAR
	VAR
		Internal	:HCRs_Cont_p_Internal_typ;
		PID	:HCRPID;
		vyServo	:HCRvyServo;
	END_VAR
END_FUNCTION_BLOCK
FUNCTION_BLOCK HCRAutoTune (* Autotuning-algorithm for Kp. *)
	VAR_INPUT
		enable	:BOOL;
		pSupply_max	:REAL;
		A_Cyl_pos	:REAL;
		A_Cyl_neg	:REAL;
		Qnom_pos	:REAL;
		Qnom_neg	:REAL;
		pDelta_nom	:REAL;
		V0_pos	:REAL;
		V0_neg	:REAL;
		h_Cyl	:REAL;
		m_Cyl	:REAL;
		s_min	:REAL;
		s_max	:REAL;
		Update	:USINT;
	END_VAR
	VAR_OUTPUT
		Kp	:REAL;
		status	:UINT;
	END_VAR
	VAR
		Internal	:HCRAutoTune_Internal_typ;
	END_VAR
END_FUNCTION_BLOCK
FUNCTION_BLOCK HCRRampGen (* Ramp generator. *)
	VAR_INPUT
		enable	:BOOL;
		t_rise	:REAL;
		t_hold	:REAL;
		t_fall	:REAL;
		y_start	:REAL;
		y_hold	:REAL;
		y_end	:REAL;
		Init	:BOOL;
	END_VAR
	VAR_OUTPUT
		y	:REAL;
		dy	:REAL;
		Finished	:BOOL;
		status	:UINT;
	END_VAR
	VAR
		Internal	:HCRRampGen_Internal_typ;
	END_VAR
END_FUNCTION_BLOCK
FUNCTION_BLOCK HCRPT1 (* 1st order delay element. *)
	VAR_INPUT
		enable	:BOOL;
		V	:REAL;
		T1	:REAL;
		u	:REAL;
		Set_y	:USINT;
		y_set	:REAL;
	END_VAR
	VAR_OUTPUT
		y	:REAL;
		status	:UINT;
	END_VAR
	VAR
		Internal	:HCRPT1_Internal_typ;
	END_VAR
END_FUNCTION_BLOCK
FUNCTION_BLOCK HCRDT1 (* 1st order differentiator. *)
	VAR_INPUT
		enable	:BOOL;
		Tv	:REAL;
		Tf	:REAL;
		u	:REAL;
		n_Avg	:USINT;
		Reset_y	:USINT;
	END_VAR
	VAR_OUTPUT
		y	:REAL;
		status	:UINT;
	END_VAR
	VAR
		Internal	:HCRDT1_Internal_typ;
	END_VAR
END_FUNCTION_BLOCK
FUNCTION_BLOCK HCRLinSpline (* Linear spline function. *)
	VAR_INPUT
		enable	:BOOL;
		NbNodes	:UINT;
		pNodeVec	:REFERENCE TO HCRNode_typ;
		Invert	:BOOL;
		Smooth	:USINT;
		Rness	:REAL;
		Update	:BOOL;
		DisMode	:SINT;
		x	:REAL;
	END_VAR
	VAR_OUTPUT
		y	:REAL;
		status	:UINT;
	END_VAR
	VAR
		Internal	:HCRLinSpline_Internal_typ;
	END_VAR
END_FUNCTION_BLOCK
FUNCTION_BLOCK HCRsF_Cont (* Switchable position/force controller (force). *)
	VAR_INPUT
		enable	:BOOL;
		pSystem_Para	:REFERENCE TO HCRSystemPara_typ;
		pValve_Para	:REFERENCE TO HCRValvePara_typ;
		pPID_Para_s	:REFERENCE TO HCRPIDPara_s_typ;
		pPID_Para_F	:REFERENCE TO HCRPIDPara_F_typ;
		vyServoMode	:USINT;
		FyServoMode	:USINT;
		tSwitch	:REAL;
		Update	:USINT;
		s_set	:REAL;
		s_act	:REAL;
		s_Cont_InVar	:HCRs_Cont_InVar_typ;
		Fp_set	:REAL;
		Fp_act	:REAL;
		F_Cont_InVar	:HCRF_Cont_InVar_typ;
		CTRLmode	:USINT;
		uSwitch	:USINT;
	END_VAR
	VAR_OUTPUT
		Qy_s	:REAL;
		Qy_Oset_s	:REAL;
		Qy_F	:REAL;
		Qy_Oset_F	:REAL;
		Qy	:REAL;
		yValve	:REAL;
		MoveDir	:SINT;
		status	:UINT;
	END_VAR
	VAR
		Internal	:HCRsF_Cont_Internal_typ;
		s_Cont	:HCRs_Cont;
		F_Cont	:HCRF_Cont;
		JoltFree	:HCRJoltFree;
	END_VAR
END_FUNCTION_BLOCK
FUNCTION_BLOCK HCRvyServo_Fp (* v-y servo correction (force). *)
	VAR_INPUT
		enable	:BOOL;
		pSupply_max	:REAL;
		pSupply	:REAL;
		pTank	:REAL;
		A_Cyl_pos	:REAL;
		A_Cyl_neg	:REAL;
		Qnom_pos	:REAL;
		Qnom_neg	:REAL;
		pDelta_nom	:REAL;
		yValve_0	:REAL;
		yValve_min	:REAL;
		Neg_y	:BOOL;
		Update	:USINT;
		Fp_Cyl	:REAL;
		Ff_Cyl_pos	:REAL;
		Ff_Cyl_neg	:REAL;
		vCyl_abs	:REAL;
		vCyl_rel	:REAL;
		Zero_yValve	:BOOL;
	END_VAR
	VAR_OUTPUT
		Qy	:REAL;
		yValve	:REAL;
		MoveDir	:SINT;
		status	:UINT;
	END_VAR
	VAR
		Internal	:HCRvyServo_Fp_Internal_typ;
	END_VAR
END_FUNCTION_BLOCK
FUNCTION_BLOCK HCRvyServo (* v-y servo correction (pressure). *)
	VAR_INPUT
		enable	:BOOL;
		pSupply_max	:REAL;
		pSupply	:REAL;
		pTank	:REAL;
		A_Cyl_pos	:REAL;
		A_Cyl_neg	:REAL;
		Qnom_pos	:REAL;
		Qnom_neg	:REAL;
		pDelta_nom	:REAL;
		yValve_0	:REAL;
		yValve_min	:REAL;
		Neg_y	:BOOL;
		Update	:USINT;
		pCyl_pos	:REAL;
		pCyl_neg	:REAL;
		vCyl_abs	:REAL;
		vCyl_rel	:REAL;
		Zero_yValve	:BOOL;
	END_VAR
	VAR_OUTPUT
		Qy	:REAL;
		yValve	:REAL;
		MoveDir	:SINT;
		status	:UINT;
	END_VAR
	VAR
		Internal	:HCRvyServo_Internal_typ;
	END_VAR
END_FUNCTION_BLOCK
FUNCTION_BLOCK HCRPID (* PID controller. *)
	VAR_INPUT
		enable	:BOOL;
		Parameter	:HCRPIDPara_typ;
		Update	:USINT;
		W	:REAL;
		X	:REAL;
		Invert	:BOOL;
		I_Switch	:SINT;
		CTRLmode	:USINT;
		Yman	:REAL;
		Yadd	:REAL;
	END_VAR
	VAR_OUTPUT
		e	:REAL;
		Yp	:REAL;
		Yi	:REAL;
		Yd	:REAL;
		Y	:REAL;
		status	:UINT;
	END_VAR
	VAR
		Internal	:HCRPID_Internal_typ;
	END_VAR
END_FUNCTION_BLOCK
FUNCTION_BLOCK HCRIT1 (* 1st order integrator. *)
	VAR_INPUT
		enable	:BOOL;
		V	:REAL;
		Tn	:REAL;
		T1	:REAL;
		u	:REAL;
		Set_y	:USINT;
		y_set	:REAL;
	END_VAR
	VAR_OUTPUT
		y	:REAL;
		status	:UINT;
	END_VAR
	VAR
		Internal	:HCRIT1_Internal_typ;
	END_VAR
END_FUNCTION_BLOCK
FUNCTION_BLOCK HCROmega0 (* Omega0-correction for Kp. *)
	VAR_INPUT
		enable	:BOOL;
		A_Cyl_pos	:REAL;
		A_Cyl_neg	:REAL;
		V0_pos	:REAL;
		V0_neg	:REAL;
		h_Cyl	:REAL;
		x_Cyl_min	:REAL;
		x_Cyl_max	:REAL;
		Update	:USINT;
		x_Cyl	:REAL;
	END_VAR
	VAR_OUTPUT
		x0_Cyl	:REAL;
		Kp_xCorr	:REAL;
		status	:UINT;
	END_VAR
	VAR
		Internal	:HCROmega0_Internal_typ;
	END_VAR
END_FUNCTION_BLOCK
FUNCTION_BLOCK HCRP2P_Cont (* Point-to-point position controller. *)
	VAR_INPUT
		enable	:BOOL;
		s_set	:REAL;
		s_act	:REAL;
		Kp	:REAL;
		P2Pmode	:SINT;
		pAddPar	:REFERENCE TO HCRP2P_Cont_AddPar_typ;
	END_VAR
	VAR_OUTPUT
		Y_P2P	:REAL;
		Y_P2P_int	:INT;
		status	:UINT;
	END_VAR
	VAR
		Internal	:HCRP2P_Cont_Internal_typ;
		PID	:HCRPID;
	END_VAR
END_FUNCTION_BLOCK
FUNCTION_BLOCK HCRF_Cont_p (* Force controller (pressure). *)
	VAR_INPUT
		enable	:BOOL;
		pSystem_Para	:REFERENCE TO HCRSystemPara_typ;
		pSystem_ParaAdd	:REFERENCE TO HCRSystemParaAdd_typ;
		pValve_Para	:REFERENCE TO HCRValvePara_typ;
		pPID_Para_F	:REFERENCE TO HCRPIDPara_F_typ;
		FyServoMode	:USINT;
		Update	:USINT;
		Fp_set	:REAL;
		Fp_act	:REAL;
		Invert	:BOOL;
		I_Switch	:USINT;
		CTRLmode	:USINT;
		Q_man	:REAL;
		Q_add	:REAL;
		dFp_set	:REAL;
		x_Cyl	:REAL;
		v_Cyl	:REAL;
		pCyl_pos	:REAL;
		pCyl_neg	:REAL;
		v_act	:REAL;
		Qy_Oset_ext	:REAL;
		Oset_Mode	:USINT;
	END_VAR
	VAR_OUTPUT
		Qy_F	:REAL;
		Qy_Oset_F	:REAL;
		Qy	:REAL;
		yValve	:REAL;
		status	:UINT;
	END_VAR
	VAR
		Internal	:HCRF_Cont_p_Internal_typ;
		PID	:HCRPID;
		FyServo	:HCRFyServo;
	END_VAR
END_FUNCTION_BLOCK
FUNCTION_BLOCK HCRPT2 (* 2nd order delay element. *)
	VAR_INPUT
		enable	:BOOL;
		V	:REAL;
		T1	:REAL;
		T2	:REAL;
		u	:REAL;
		Set_y	:USINT;
		y_set	:REAL;
	END_VAR
	VAR_OUTPUT
		y	:REAL;
		status	:UINT;
	END_VAR
	VAR
		Internal	:HCRPT2_Internal_typ;
	END_VAR
END_FUNCTION_BLOCK
FUNCTION_BLOCK HCRPT2s (* Oscillating 2nd order delay element. *)
	VAR_INPUT
		enable	:BOOL;
		V	:REAL;
		D	:REAL;
		Tf	:REAL;
		u	:REAL;
		Set_y	:USINT;
		y_set	:REAL;
	END_VAR
	VAR_OUTPUT
		y	:REAL;
		status	:UINT;
	END_VAR
	VAR
		Internal	:HCRPT2s_Internal_typ;
	END_VAR
END_FUNCTION_BLOCK
FUNCTION_BLOCK HCRDT2s (* Oscillating 2nd order differentiator. *)
	VAR_INPUT
		enable	:BOOL;
		D	:REAL;
		Tv	:REAL;
		Tf	:REAL;
		u	:REAL;
		Reset_y	:USINT;
	END_VAR
	VAR_OUTPUT
		y	:REAL;
		status	:UINT;
	END_VAR
	VAR
		Internal	:HCRDT2s_Internal_typ;
	END_VAR
END_FUNCTION_BLOCK
FUNCTION_BLOCK HCRPT1cP (* Converging 1st order delay element. *)
	VAR_INPUT
		enable	:BOOL;
		T1	:REAL;
		u	:REAL;
		Set_y	:USINT;
		y_set	:REAL;
	END_VAR
	VAR_OUTPUT
		y	:REAL;
		status	:UINT;
	END_VAR
	VAR
		Internal	:HCRPT1cP_Internal_typ;
	END_VAR
END_FUNCTION_BLOCK
FUNCTION_BLOCK HCRJoltFree (* Jolt-free switching between 2 inputs. *)
	VAR_INPUT
		enable	:BOOL;
		tSwitch	:REAL;
		uSwitch	:BOOL;
		u1	:REAL;
		u2	:REAL;
	END_VAR
	VAR_OUTPUT
		y	:REAL;
		status	:UINT;
	END_VAR
	VAR
		Internal	:HCRJoltFree_Internal_typ;
		PT1cP	:HCRPT1cP;
	END_VAR
END_FUNCTION_BLOCK
FUNCTION_BLOCK HCRLinValve (* Valve linearization. *)
	VAR_INPUT
		enable	:BOOL;
		NbNodes	:UINT;
		pNodeVec	:REFERENCE TO HCRNode_typ;
		Neg_Uy	:BOOL;
		Update	:BOOL;
		DisMode	:SINT;
		Qy	:REAL;
	END_VAR
	VAR_OUTPUT
		Uy	:REAL;
		status	:UINT;
	END_VAR
	VAR
		Internal	:HCRLinValve_Internal_typ;
		LinSpline	:HCRLinSpline;
	END_VAR
END_FUNCTION_BLOCK
FUNCTION_BLOCK HCRF_Cont (* Force controller (force). *)
	VAR_INPUT
		enable	:BOOL;
		pSystem_Para	:REFERENCE TO HCRSystemPara_typ;
		pValve_Para	:REFERENCE TO HCRValvePara_typ;
		pPID_Para_F	:REFERENCE TO HCRPIDPara_F_typ;
		FyServoMode	:USINT;
		Update	:USINT;
		Fp_set	:REAL;
		Fp_act	:REAL;
		Invert	:BOOL;
		I_Switch	:USINT;
		CTRLmode	:USINT;
		Q_man	:REAL;
		Q_add	:REAL;
		v_act	:REAL;
		Qy_Oset_ext	:REAL;
		Oset_Mode	:USINT;
	END_VAR
	VAR_OUTPUT
		Qy_F	:REAL;
		Qy_Oset_F	:REAL;
		Qy	:REAL;
		yValve	:REAL;
		status	:UINT;
	END_VAR
	VAR
		Internal	:HCRF_Cont_Internal_typ;
		PID	:HCRPID;
		FyServo_Fp	:HCRFyServo_Fp;
	END_VAR
END_FUNCTION_BLOCK
FUNCTION_BLOCK HCRs_Cont (* Position controller (force). *)
	VAR_INPUT
		enable	:BOOL;
		pSystem_Para	:REFERENCE TO HCRSystemPara_typ;
		pValve_Para	:REFERENCE TO HCRValvePara_typ;
		pPID_Para_s	:REFERENCE TO HCRPIDPara_s_typ;
		vyServoMode	:USINT;
		Update	:USINT;
		s_set	:REAL;
		s_act	:REAL;
		Invert	:BOOL;
		I_Switch	:USINT;
		CTRLmode	:USINT;
		v_man	:REAL;
		v_add	:REAL;
		v_set	:REAL;
		Fp_Cyl	:REAL;
		Ff_Cyl_pos	:REAL;
		Ff_Cyl_neg	:REAL;
		Qy_Oset_ext	:REAL;
		Oset_Mode	:USINT;
	END_VAR
	VAR_OUTPUT
		Qy_s	:REAL;
		Qy_Oset_s	:REAL;
		Qy	:REAL;
		yValve	:REAL;
		MoveDir	:SINT;
		status	:UINT;
	END_VAR
	VAR
		Internal	:HCRs_Cont_Internal_typ;
		PID	:HCRPID;
		vyServo_Fp	:HCRvyServo_Fp;
	END_VAR
END_FUNCTION_BLOCK
FUNCTION_BLOCK HCRSPF (* Smart path finder. *)
	VAR_INPUT
		enable	:BOOL;
		pMove_Para	:REFERENCE TO HCRMovePara_typ;
		Stop	:BOOL;
		s_home	:REAL;
		Set_home	:BOOL;
		s_end	:REAL;
		Init	:BOOL;
		Brake	:BOOL;
	END_VAR
	VAR_OUTPUT
		s_set	:REAL;
		v_set	:REAL;
		a_set	:REAL;
		MoveDir	:SINT;
		ApproachDir	:SINT;
		Reached	:BOOL;
		status	:UINT;
	END_VAR
	VAR
		Internal	:HCRSPF_Internal_typ;
		SystemInfo	:SysInfo;
	END_VAR
END_FUNCTION_BLOCK
FUNCTION_BLOCK HCRFyServo_Fp (* F-y servo correction (force). *)
	VAR_INPUT
		enable	:BOOL;
		pSupply_max	:REAL;
		pSupply	:REAL;
		pTank	:REAL;
		A_Cyl_pos	:REAL;
		A_Cyl_neg	:REAL;
		Qnom_pos	:REAL;
		Qnom_neg	:REAL;
		Neg_y	:BOOL;
		Update	:USINT;
		Fp	:REAL;
		u	:REAL;
	END_VAR
	VAR_OUTPUT
		Qy	:REAL;
		yValve	:REAL;
		status	:UINT;
	END_VAR
	VAR
		Internal	:HCRFyServo_Fp_Internal_typ;
	END_VAR
END_FUNCTION_BLOCK
FUNCTION_BLOCK HCRFIFO (* FIFO (dead time) element. *)
	VAR_INPUT
		enable	:BOOL;
		t_FIFO	:DINT;
		x	:REAL;
		Set_y	:BOOL;
		y_set	:REAL;
	END_VAR
	VAR_OUTPUT
		y	:REAL;
		status	:UINT;
	END_VAR
	VAR
		Internal	:HCRFIFO_Internal_typ;
	END_VAR
END_FUNCTION_BLOCK
FUNCTION_BLOCK HCRDT2 (* 2nd order differentiator. *)
	VAR_INPUT
		enable	:BOOL;
		Tv	:REAL;
		T1	:REAL;
		T2	:REAL;
		u	:REAL;
		n_Avg	:USINT;
		Reset_y	:USINT;
	END_VAR
	VAR_OUTPUT
		y	:REAL;
		status	:UINT;
	END_VAR
	VAR
		Internal	:HCRDT2_Internal_typ;
	END_VAR
END_FUNCTION_BLOCK
FUNCTION_BLOCK HCRSFG (* Smart force generator. *)
	VAR_INPUT
		enable	:BOOL;
		t_Jolt	:REAL;
		Stop	:BOOL;
		dFp_home	:REAL;
		Fp_home	:REAL;
		Set_home	:BOOL;
		t_delta	:REAL;
		Fp_end	:REAL;
		Init	:BOOL;
	END_VAR
	VAR_OUTPUT
		Fp_set	:REAL;
		dFp_set	:REAL;
		t_delta_act	:REAL;
		Reached	:BOOL;
		status	:UINT;
	END_VAR
	VAR
		Internal	:HCRSFG_Internal_typ;
		SPF	:HCRSPF;
	END_VAR
END_FUNCTION_BLOCK
FUNCTION_BLOCK HCRFyServo (* F-y servo correction (pressure). *)
	VAR_INPUT
		enable	:BOOL;
		pSupply_max	:REAL;
		pSupply	:REAL;
		pTank	:REAL;
		A_Cyl_pos	:REAL;
		A_Cyl_neg	:REAL;
		Qnom_pos	:REAL;
		Qnom_neg	:REAL;
		pDelta_nom	:REAL;
		V0_pos	:REAL;
		V0_neg	:REAL;
		h_Cyl	:REAL;
		Neg_y	:BOOL;
		Update	:USINT;
		x_Cyl	:REAL;
		v_Cyl	:REAL;
		pCyl_pos	:REAL;
		pCyl_neg	:REAL;
		dF_Cyl_abs	:REAL;
		dF_Cyl_rel	:REAL;
	END_VAR
	VAR_OUTPUT
		Qy	:REAL;
		yValve	:REAL;
		status	:UINT;
	END_VAR
	VAR
		Internal	:HCRFyServo_Internal_typ;
	END_VAR
END_FUNCTION_BLOCK

(* ---- AsHydCon.var ---- *)
VAR CONSTANT
	HCR_ERR_SPF_A_DEC_POS_NEG_ZERO	: UINT	:= 32292;
	HCR_ERR_SPF_A_DEC_NEG_NEG_ZERO	: UINT	:= 32291;
	HCR_ERR_SPF_A_ACC_POS_NEG_ZERO	: UINT	:= 32290;
	HCR_ERR_SPF_A_ACC_NEG_NEG_ZERO	: UINT	:= 32289;
	HCR_WARN_SERVO_P_CYL_POS_HIGH	: UINT	:= 32407;
	HCR_WARN_SERVO_P_CYL_NEG_HIGH	: UINT	:= 32404;
	HCR_WARN_LIN_Y_NOT_ASC_DESC_S	: UINT	:= 32385;
	HCR_WARN_LIN_X_NOT_ASC_DESC_S	: UINT	:= 32383;
	HCR_WARN_SERVO_P_CYL_POS_NEG	: UINT	:= 32409;
	HCR_WARN_SERVO_P_CYL_POS_LOW	: UINT	:= 32408;
	HCR_WARN_SERVO_P_CYL_NEG_NEG	: UINT	:= 32406;
	HCR_WARN_SERVO_P_CYL_NEG_LOW	: UINT	:= 32405;
	HCR_WARN_AUTOTUNE_KP_INVALID	: UINT	:= 32413;
	HCR_ERR_SPF_PER_S_PERIOD_NEG	: UINT	:= 32312;
	HCR_ERR_SFG_T_DELTA_NEG_ZERO	: UINT	:= 32315;
	HCR_ERR_OMEGA0_X_CYL_MIN_MAX	: UINT	:= 32310;
	HCR_WARN_LIN_Y_NOT_ASC_DESC	: UINT	:= 32384;
	HCR_WARN_JFREE_TSWITCH_ZERO	: UINT	:= 32380;
	HCR_ERR_SYSTEM_P_SUPPLY_MAX	: UINT	:= 32300;
	HCR_ERR_SPF_VC_POS_NEG_ZERO	: UINT	:= 32296;
	HCR_ERR_SPF_VC_NEG_NEG_ZERO	: UINT	:= 32295;
	HCR_WARN_JFREE_TSWITCH_5TS	: UINT	:= 32379;
	HCR_ERR_PID_D_MODE_INVALID	: UINT	:= 32263;
	HCR_ERR_LIN_Y_NOT_ASC_DESC	: UINT	:= 32261;
	HCR_ERR_LIN_X_NOT_ASC_DESC	: UINT	:= 32260;
	HCR_WARN_SERVO_FF_CYL_POS	: UINT	:= 32403;
	HCR_WARN_SERVO_FF_CYL_NEG	: UINT	:= 32402;
	HCR_ERR_VALVE_P_DELTA_NOM	: UINT	:= 32283;
	HCR_ERR_NOTCH_F0_NEG_ZERO	: UINT	:= 32308;
	HCR_ERR_LIN_NODEVEC_EMPTY	: UINT	:= 32259;
	HCR_ERR_JFREE_TSWITCH_NEG	: UINT	:= 32258;
	HCR_ERR_DT12S_TF_NEG_ZERO	: UINT	:= 32254;
	HCR_WARN_SFG_T_DELTA_ACT	: UINT	:= 32420;
	HCR_WARN_SERVO_V_CYL_MAX	: UINT	:= 32410;
	HCR_WARN_FIFO_T_FIFO_INT	: UINT	:= 32377;
	HCR_ERR_PT2S_TF_NEG_ZERO	: UINT	:= 32277;
	HCR_ERR_NOTCH_B_NEG_ZERO	: UINT	:= 32307;
	HCR_ERR_DT12S_T1_T2_ZERO	: UINT	:= 32252;
	HCR_WARN_LIN_CRIT_RNESS	: UINT	:= 32381;
	HCR_WARN_FIFO_T_FIFO_TS	: UINT	:= 32378;
	HCR_ERR_SYSTEM_P_SUPPLY	: UINT	:= 32281;
	HCR_ERR_RAMP_T_RISE_NEG	: UINT	:= 32288;
	HCR_ERR_RAMP_T_HOLD_NEG	: UINT	:= 32287;
	HCR_ERR_RAMP_T_FALL_NEG	: UINT	:= 32286;
	HCR_ERR_IT1_TN_NEG_ZERO	: UINT	:= 32314;
	HCR_ERR_FIFO_T_FIFO_NEG	: UINT	:= 32257;
	HCR_WARN_SPF_PER_S_END	: UINT	:= 32415;
	HCR_WARN_PT1CP_T1_ZERO	: UINT	:= 32400;
	HCR_WARN_PID_TN_POS_TS	: UINT	:= 32388;
	HCR_WARN_PID_TN_NEG_TS	: UINT	:= 32387;
	HCR_WARN_DT12S_TV_ZERO	: UINT	:= 32376;
	HCR_WARN_DT12S_T2_ZERO	: UINT	:= 32373;
	HCR_WARN_DT12S_T1_ZERO	: UINT	:= 32371;
	HCR_ERR_SYSTEM_NIL_PTR	: UINT	:= 32299;
	HCR_ERR_SPF_VC_POS_NEG	: UINT	:= 32296;
	HCR_ERR_SPF_VC_NEG_NEG	: UINT	:= 32295;
	HCR_ERR_SPF_T_JOLT_NEG	: UINT	:= 32294;
	HCR_ERR_SPF_PER_S_HOME	: UINT	:= 32311;
	HCR_ERR_SFG_T_JOLT_NEG	: UINT	:= 32317;
	HCR_ERR_PID_WX_MAX_MIN	: UINT	:= 32271;
	HCR_ERR_PID_TN_POS_NEG	: UINT	:= 32269;
	HCR_ERR_PID_TN_NEG_NEG	: UINT	:= 32268;
	HCR_ERR_PID_DY_MAX_NEG	: UINT	:= 32262;
	HCR_WARN_PT12_T2_ZERO	: UINT	:= 32398;
	HCR_WARN_PT12_T1_ZERO	: UINT	:= 32396;
	HCR_WARN_PID_YMAN_MIN	: UINT	:= 32394;
	HCR_WARN_PID_YMAN_MAX	: UINT	:= 32393;
	HCR_WARN_PID_YADD_100	: UINT	:= 32390;
	HCR_ERR_VALVE_NIL_PTR	: UINT	:= 32306;
	HCR_ERR_SYSTEM_V0_POS	: UINT	:= 32302;
	HCR_ERR_SYSTEM_V0_NEG	: UINT	:= 32301;
	HCR_ERR_SYSTEM_P_TANK	: UINT	:= 32282;
	HCR_ERR_SYSTEM_P_DIFF	: UINT	:= 32280;
	HCR_ERR_SERVO_MODE_VY	: UINT	:= 32304;
	HCR_ERR_SERVO_MODE_FY	: UINT	:= 32303;
	HCR_ERR_PID_Y_MAX_MIN	: UINT	:= 32272;
	HCR_ERR_PID_K_FBK_NEG	: UINT	:= 32265;
	HCR_ERR_OMEGA0_X0_CYL	: UINT	:= 32309;
	HCR_WARN_SERVO_Y_MAX	: UINT	:= 32411;
	HCR_WARN_PT1CP_T1_TS	: UINT	:= 32399;
	HCR_WARN_NOTCH_F0_FS	: UINT	:= 32414;
	HCR_WARN_LIN_NB_NODE	: UINT	:= 32382;
	HCR_WARN_IT1_T1_ZERO	: UINT	:= 32417;
	HCR_WARN_DT12S_TV_TS	: UINT	:= 32375;
	HCR_WARN_DT12S_TF_TS	: UINT	:= 32374;
	HCR_WARN_DT12S_T2_TS	: UINT	:= 32372;
	HCR_WARN_DT12S_T1_TS	: UINT	:= 32370;
	HCR_ERR_SYSTEM_M_CYL	: UINT	:= 32298;
	HCR_ERR_SYSTEM_H_CYL	: UINT	:= 32297;
	HCR_ERR_SYSTEM_A_CYL	: UINT	:= 32279;
	HCR_ERR_PT1CP_T1_NEG	: UINT	:= 32275;
	HCR_ERR_DT12S_TV_NEG	: UINT	:= 32255;
	HCR_ERR_DT12S_T2_NEG	: UINT	:= 32253;
	HCR_ERR_DT12S_T1_NEG	: UINT	:= 32251;
	HCR_WARN_SFG_FP_END	: UINT	:= 32419;
	HCR_WARN_PT2S_TF_TS	: UINT	:= 32401;
	HCR_WARN_PT12_T2_TS	: UINT	:= 32397;
	HCR_WARN_PT12_T1_TS	: UINT	:= 32395;
	HCR_WARN_PID_YI_MIN	: UINT	:= 32392;
	HCR_WARN_PID_YI_MAX	: UINT	:= 32391;
	HCR_ERR_VALVE_Q_NOM	: UINT	:= 32284;
	HCR_ERR_SPF_NIL_PTR	: UINT	:= 32293;
	HCR_ERR_SERVO_Y_MIN	: UINT	:= 32278;
	HCR_ERR_PT12_T2_NEG	: UINT	:= 32274;
	HCR_ERR_PT12_T1_NEG	: UINT	:= 32273;
	HCR_ERR_PID_TF_ZERO	: UINT	:= 32267;
	HCR_ERR_PID_NIL_PTR	: UINT	:= 32305;
	HCR_ERR_DT12S_D_NEG	: UINT	:= 32250;
	HCR_WARN_PID_TV_TS	: UINT	:= 32389;
	HCR_WARN_PID_TF_TS	: UINT	:= 32386;
	HCR_WARN_IT1_TN_TS	: UINT	:= 32418;
	HCR_WARN_IT1_T1_TS	: UINT	:= 32416;
	HCR_ERR_SFG_T_DIFF	: UINT	:= 32316;
	HCR_ERR_PT2S_D_NEG	: UINT	:= 32276;
	HCR_ERR_PID_TV_NEG	: UINT	:= 32270;
	HCR_ERR_PID_TF_NEG	: UINT	:= 32266;
	HCR_ERR_PID_KW_0_1	: UINT	:= 32264;
	HCR_ERR_IT1_T1_NEG	: UINT	:= 32313;
	HCR_ERR_VALVE_Y_0	: UINT	:= 32285;
	HCR_WARN_SPF_MEM	: UINT	:= 32412;
	HCR_ERR_FIFO_MEM	: UINT	:= 32256;
	HCR_ERR_DISABLED	: UINT	:= 65534;
END_VAR
